FUNCTION_BLOCK FB_CC_TempSensorTest EXTENDS FB_TestSuite
VAR
    fbTempSensor: FB_CC_TempSensor;
    fbFFHWO: FB_HardwareFFOutput;
END_VAR


TestBasic();
TestThresholdVeto();
TestAutoReset();

METHOD SetTempAndRunFB
VAR_INPUT
    iRawTemp: INT;
END_VAR
VAR
    ptr: POINTER TO INT;
END_VAR

ptr := ADR(fbTempSensor.iRaw);
ptr^ := iRawTemp * 10;

fbTempSensor(io_fbFFHWO:=fbFFHWO);
fbFFHWO.ExecuteNoLog();
END_METHOD

METHOD TestAutoReset
VAR_INPUT
END_VAR

TEST('TestAutoReset');

// Set a fixed threshold for the test
fbTempSensor.fFaultThreshold := 30;

// Clear faults
fbTempSensor.bVeto := TRUE;
SetTempAndRunFB(0);
AssertTrue(
    fbFFHWO.astFF[fbTempSensor.FFO.RegistrationIdx].BeamPermitted,
    'Beam not permitted after full clear with low temp',
);

// Cause a fault
fbTempSensor.bVeto := FALSE;
SetTempAndRunFB(100);
AssertFalse(
    fbFFHWO.astFF[fbTempSensor.FFO.RegistrationIdx].BeamPermitted,
    'Beam permitted after high temp',
);

// Remove the fault condition, should still be fauling
fbTempSensor.bVeto := FALSE;
SetTempAndRunFB(0);
AssertFalse(
    fbFFHWO.astFF[fbTempSensor.FFO.RegistrationIdx].BeamPermitted,
    'Beam permitted before manual reset',
);

// Set veto, should no longer be faulting
fbTempSensor.bVeto := TRUE;
SetTempAndRunFB(0);
AssertTrue(
    fbFFHWO.astFF[fbTempSensor.FFO.RegistrationIdx].BeamPermitted,
    'Beam not permitted after veto',
);

TEST_FINISHED();
END_METHOD

METHOD TestBasic

TEST('TestBasic');

fbTempSensor.fFaultThreshold := 10;
fbTempSensor.bVeto := FALSE;
SetTempAndRunFB(2);
AssertTrue(
    fbTempSensor.FFO.i_xOK,
    'Faulted with temp below threshold',
);

fbTempSensor.fFaultThreshold := 10;
fbTempSensor.bVeto := FALSE;
SetTempAndRunFB(150);
AssertFalse(
    fbTempSensor.FFO.i_xOK,
    'Did not fault with temp above threshold',
);

fbTempSensor.fFaultThreshold := 5;
fbTempSensor.bVeto := TRUE;
SetTempAndRunFB(1000);
AssertTrue(
    fbTempSensor.FFO.i_xOK,
    'Faulted with manual veto',
);

TEST_FINISHED();
END_METHOD

METHOD TestThresholdVeto

TEST('TestThresholdVeto');

fbTempSensor.fFaultThreshold := 0;
fbTempSensor.bVeto := FALSE;
SetTempAndRunFB(500);
AssertTrue(
    fbTempSensor.FFO.i_xOK,
    'Faulted with not-loaded threshold',
);

TEST_FINISHED();
END_METHOD

END_FUNCTION_BLOCK

(* stored: Version 1.1.0.1
   POU FB_CC_TempSensorTest: Id {97eee846-433c-4b59-96d7-8ed3430964de}, SpecialFunc None
   Method SetTempAndRunFB: Id {31ab1f78-a5de-4c4f-b101-c9bfbb785b79}
   Method TestAutoReset: Id {9b135c6c-5fae-4bb3-aa3c-5e9e36ae077f}
   Method TestBasic: Id {dcdef24a-9782-4bfe-88f4-1b54e4b20aed}
   Method TestThresholdVeto: Id {e88f0c37-f17e-4f5e-9576-320395957b83} *)
